{attribute addProperty BoxType "EK1100-0000-0018"}
{attribute addProperty Id "Beckhoff_EP7xxxEK1122Beckhoff_EP7xxxEK1122_A7CCCB3C142491781.125"}
{attribute addProperty CRC "1530051452"}
{attribute addProperty SizeInBites "14249"}
{attribute addProperty SizeInBytes "1781.125"}
TYPE Beckhoff_EP7xxx_5B32BB7C EXTENDS EK1100_179A0949 :
STRUCT
	{attribute addProperty Name "Beckhoff_EP7xxxEK1122"}
	Beckhoff_EP7xxxEK1122 : Beckhoff_EP7xxxEK1122_A7CCCB3C;
END_STRUCT
END_TYPE

(* stored: Version 1.2.0.0, ProductVersion 3.1.4024.9
   DUT Beckhoff_EP7xxx_5B32BB7C: Id {f56deaaf-69f0-4b24-aa6d-ab64dafc224a} *)
